(* CoDeSys 2.3 export: STANDBY.EXP *)

(* POU Initialisation_Standby/StandBY, SFC *)
PROGRAM StandBY
VAR
END_VAR
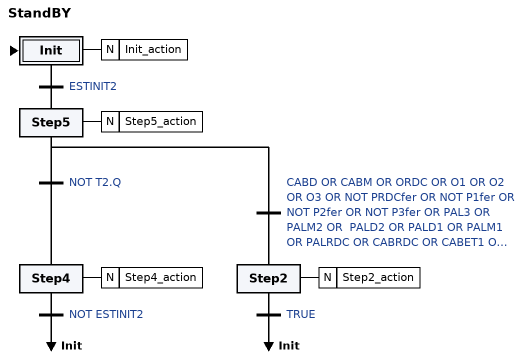
INITIAL_STEP Init:
	Init_action(N);
END_STEP
TRANSITION FROM Init TO Step5 := ESTINIT2;
END_TRANSITION
STEP Step5:
	Step5_action(N);
END_STEP
TRANSITION FROM Step5 TO Step4 := NOT T2.Q;
END_TRANSITION
TRANSITION FROM Step5 TO Step2 := CABD OR CABM OR ORDC OR O1 OR O2 OR O3 OR NOT PRDCfer OR NOT P1fer OR NOT P2fer OR NOT P3fer OR PAL3 OR PALM2 OR  PALD2 OR PALD1 OR PALM1 OR PALRDC OR CABRDC OR CABET1 OR CABET2 OR CABET3;
END_TRANSITION
STEP Step4:
	Step4_action(N);
END_STEP
TRANSITION FROM Step4 TO Init := NOT ESTINIT2;
END_TRANSITION
STEP Step2:
	Step2_action(N);
END_STEP
TRANSITION FROM Step2 TO Init := TRUE;
END_TRANSITION

ACTION Init_action:
T2(IN:=FALSE);
END_ACTION

ACTION Step5_action:
T2(IN:=TRUE, PT:=t#7s);
END_ACTION

ACTION Step4_action:
T2(IN:=FALSE);
ESTINIT2:=FALSE;
StanbyActive:=TRUE;
END_ACTION

ACTION Step2_action:
(* IF  CABD OR CABM OR ORDC OR O1 OR O2 OR O3 OR NOT PRDCfer OR NOT P1fer OR NOT P2fer OR NOT P3fer OR PAL3 OR PALM2 OR  PALD2 OR PALD1 OR PALM1 OR PALRDC THEN
	T2(IN:=TRUE, PT:=t#10s);
ELSE
	T2(IN:=FALSE);
END_IF
*)

T2(IN:=FALSE);
T2(IN:=TRUE, PT:=t#1ms);
END_ACTION
END_PROGRAM
